INTERFACE I_LimSwStatus

METHOD AxisStatus
VAR_INPUT
	HomeBusy: BOOL;
	PositiveDirection : BOOL;
	NegativeDirection : BOOL;
END_VAR
END_METHOD

METHOD DriveCommands
VAR_INPUT
	Enable: BOOL;
	NewMoveReq : BOOL;
	Reset: BOOL;
END_VAR
END_METHOD

PROPERTY LimBackward : BOOL
GET
END_GET
END_PROPERTY

PROPERTY LimForward : BOOL
GET
END_GET
END_PROPERTY

PROPERTY LimHit : BOOL
GET
END_GET
END_PROPERTY

PROPERTY LimHome : BOOL
GET
END_GET
END_PROPERTY

PROPERTY Message : T_MAXSTRING
GET
END_GET
END_PROPERTY

PROPERTY MoveBackwardEnabled : BOOL
GET
END_GET
END_PROPERTY

PROPERTY MoveForwardEnabled : BOOL
GET
END_GET
END_PROPERTY

PROPERTY Warning : BOOL
GET
END_GET
END_PROPERTY

END_INTERFACE

(* stored: Version 1.1.0.1
   Itf I_LimSwStatus: Id {256e382d-89de-4efb-b391-22faa6fe67b6}
   Method AxisStatus: Id {ad2a89e1-41ec-4053-88de-27c1f75c0736}
   Method DriveCommands: Id {df511f30-cad4-4303-88ab-dcbcab9d3c4d}
   Property LimBackward: Id {d3e174fe-8267-4de9-813d-46b0b3cd2d9c}
   Get Get: Id {a3b4afe5-0e5a-44af-aa9a-8370d1c91f06}
   Property LimForward: Id {4df30b89-8ee7-49f7-b129-3ca64eaa1735}
   Get Get: Id {5e40816d-8df5-4674-a88e-d1f52596914e}
   Property LimHit: Id {dee2d2af-22a0-47af-ab9b-17dc48dde618}
   Get Get: Id {fc9ea001-e8c2-4858-954a-09da4fcb8eea}
   Property LimHome: Id {f84feb6e-7376-4267-ad4f-1dd43787e440}
   Get Get: Id {19bd3ff6-6d16-4669-8dec-b80565590b18}
   Property Message: Id {e8b10816-08b9-43cf-a44e-3e2b5c9d0ccf}
   Get Get: Id {1ea16d51-c727-4125-a99b-38bd676d8335}
   Property MoveBackwardEnabled: Id {b4e7f086-2ef8-4485-be7e-4532b5db4264}
   Get Get: Id {9b0ef177-2451-44cd-bad6-e27eaa34b91b}
   Property MoveForwardEnabled: Id {c448b972-f646-4f09-a55d-f335dff878cb}
   Get Get: Id {63539f14-b019-40ce-9a44-701a06eafced}
   Property Warning: Id {1b98f41d-ef99-4e0f-8e76-a2ade70cd32d}
   Get Get: Id {25b7225f-f85c-46d5-99ff-635c5137c3d3} *)
